Fanuc KAREL source: kf00098.KL

PROGRAM KF00098
%NOLOCKGROUP
%ENVIRONMENT REGOPE
VAR
I:INTEGER;J:INTEGER;X:REAL;Y:REAL;B:BOOLEAN;C:BOOLEAN;TXT : STRING[80];TXT2 : STRING[80];AI : ARRAY[4] OF INTEGER;BI : ARRAY[4] OF INTEGER;P : XYZWPR
JP : JOINTPOS9
PF : POSITION
V1 : VECTOR
V2 : VECTOR
STATUS:INTEGER
BEGIN
--
--
--
--
--
--
--
--
--
--
I=3
X=2.5
SET_REAL_REG(1,X,STATUS)
END KF00098
